// TIA Portal V17 export
// export: Created 2026-04-13T11:12:43.2794496Z, ExportSetting WithDefaults, DisplayName Totally Integrated Automation Portal, DisplayVersion V17 Update 4, DisplayName TIA Portal Openness, DisplayVersion V17 Update 4, DisplayName TIA Portal Version Control Interface, DisplayVersion V17, DisplayName SINAMICS Startdrive Advanced, DisplayVersion V17, DisplayName SINAMICS Startdrive G130, G150, S120, S150, SINAMICS MV, S210, DisplayVersion V17, DisplayName SINAMICS Startdrive G110M, G120, G120C, G120D, G120P, G115D, DisplayVersion V17, DisplayName STEP 7 Professional, DisplayVersion V17 Update 4, DisplayName STEP 7 Safety, DisplayVersion V17, DisplayName WinCC Professional, DisplayVersion V17 Update 4
FUNCTION "随机生成数" : Void   // FC39, SCL
{ S7_Optimized_Access := 'TRUE' }
VERSION : 0.1
// stored: AutoNumber true, IsIECCheckEnabled false, SetENOAutomatically false, UDAEnableTagReadback false
   VAR_INPUT
      最小生成数 : Real;
      偏置 : Real;
      数据类型 : Bool;   // 0为实数，1为整数
   END_VAR
   VAR_OUTPUT
      随机数 : Real;
   END_VAR
BEGIN
   IF #数据类型 THEN
       #随机数 := REAL_TO_DINT(INT_TO_REAL("Clock_Byte") / 255 * #偏置 + #最小生成数);
   ELSE
       #随机数 := INT_TO_REAL("Clock_Byte") / 255 * #偏置 + #最小生成数;
   END_IF;
END_FUNCTION
